(*
SPDX-FileCopyrightText: © 2026 Oleksandr Tiutyk <trofimich@gmail.com>
SPDX-License-Identifier: MIT
License: https://opensource.org/license/mit
*)

(*!
<summary>Reports that a fixed-capacity collection cannot accept another element.</summary>
<description>
The caller detects the condition; this exception does not inspect or modify the collection or destination.
Uses the GeneralException task-local cycle lifetime and throw rules. Dynamic copies are explicitly registered
by Clone after construction; plain __NEW does not transfer ownership to the task manager.
</description>
*)

{attribute 'enable_dynamic_creation'}
{attribute 'no_explicit_call' := 'do not call this function block directly'}
FUNCTION_BLOCK StaticCollectionFullException EXTENDS GeneralException IMPLEMENTS IStaticCollectionFullException
VAR_STAT
	//! <summary>Class name shared by all instances of this function block.</summary>
	{attribute 'hide'} 
	_ClassName : STRING := __POUNAME();
END_VAR

{attribute 'monitoring' := 'call'}
PROPERTY ClassName : REFERENCE TO STRING
GET
ClassName REF= _ClassName;
END_GET
END_PROPERTY

(*!
<summary>Creates a clone of this concrete exception type.</summary>
<description>
Copies GeneralException fields and timestamps. The clone belongs to DynamicMemoryManager until cleanup of the
creating task; callers must not delete it. Allocation failure is terminal. Registers the newly constructed
instance before copying payload, outside FB_init. Registration failure releases the unregistered instance and
raises a terminal error; copy failure leaves the registered instance owned by the task manager for cleanup.
Custom overrides must follow the same ownership sequence.
</description>
*)
METHOD Clone : IObject
VAR
	exceptionClone : POINTER TO StaticCollectionFullException;
END_VAR
exceptionClone := __NEW(StaticCollectionFullException);

IF exceptionClone = 0 THEN
	DynamicMemoryManager.RaiseAllocationFailure();
END_IF

DynamicMemoryManager.RegisterAutoDisposedObject(autoDisposedObject := exceptionClone^);

exceptionClone^.CopyGeneralFields(sourceException := THIS^);

Clone := exceptionClone^;
END_METHOD

(*!
<summary>Provides the library namespace used in diagnostics.</summary>
<description>
Borrowed read-only reference to the compiler-initialized library namespace; no ownership transfer.
</description>
*)
{attribute 'monitoring' := 'call'}
PROPERTY NamespaceName : REFERENCE TO STRING
GET
NamespaceName REF= CurrentNamespace.Name;
END_GET
END_PROPERTY

(*!
<summary>Reports the byte size of this concrete instance.</summary>
<description>
Uses XSIZEOF on the instance. Does not include separately allocated payloads or prove that an arbitrary
address is valid.
</description>
*)
{attribute 'monitoring' := 'call'}
PROPERTY SelfSize : ULINT
GET
SelfSize := XSIZEOF(THIS^);
END_GET
END_PROPERTY

(*!
<summary>Builds the diagnostic and raises this exception through GeneralException.</summary>
<description>
Copies the supplied diagnostic data, sets error code to zero and supplies no inner exception. Call only in a
cyclic task, not during FB_init. The caller must already have detected the reported condition.
</description>
<param name="collectionName">Collection name used in the diagnostic.</param>
<param name="capacity">Maximum number of elements, not a byte size.</param>
*)
METHOD Throw
VAR_INPUT
	sourceNamespaceName : STRING;
	sourceClassName : STRING;
	sourcePOUName : STRING;
	sourcePosition : STRING;
	collectionName : WSTRING;
	capacity : UDINT;
END_VAR
VAR
	message : ERROR_MESSAGE;
END_VAR

message := WideStrings.Concat255(
	"Static collection '",
	collectionName,
	"' is full (capacity is ",
	TO_WSTRING(capacity),
	")"
);

InternalThrow(
	sourceNamespaceName := sourceNamespaceName,
	sourceClassName := sourceClassName,
	sourcePOUName := sourcePOUName,
	sourcePosition := sourcePosition,
	message := message,
	errorCode := 0,
	innerException := 0
);
END_METHOD

END_FUNCTION_BLOCK

(* stored: Version 1.1.0.1
   POU StaticCollectionFullException: Id {0096f1a9-f507-4fb2-a70c-f47e70fe3987}, SpecialFunc None
   Property ClassName: Id {93be92f8-bd0c-4e55-bb0c-ccc3953174b7}
   Get Get: Id {827b5504-d29b-4914-a7e3-a0d60e070fd8}
   Method Clone: Id {3441f170-2e5d-457f-b92b-797f55fe8a8b}
   Property NamespaceName: Id {22708afd-502c-463f-a9c3-de8b55baf047}
   Get Get: Id {35a686c5-79f5-4a96-bc6f-2cb3126d98ca}
   Property SelfSize: Id {25fc0a8f-780c-4fc5-97d3-463e17b3b9be}
   Get Get: Id {4c813345-d41d-4244-8ff5-68226cb89364}
   Method Throw: Id {306cfa76-a1cd-4575-8605-c209c5fbe1e7} *)
